// TIA Portal project "141db_PLcen hasera" (V15.1)

(* hardware
DEVICE "S7-1200 station_1"  S7-1200 Station
   slot 0: "Rack_0"  S7-1200 Rack  Rack  V1.0
   slot 1: "PLC_1"  CPU 1214C AC/DC/Rly  6ES7 214-1BG40-0XB0  V4.2
   slot 3: "AQ 1x12BIT_1"  AQ1 signal board  6ES7 232-4HA30-0XB0  V1.0
*)

// ===== PLC "PLC_1"  CPU 1214C AC/DC/Rly =====

VAR_GLOBAL   // PLC tag table "Tabla de variables estándar"
   "Etapa0" AT %M16.0 : Bool;
   "S1" AT %I1.0 : Bool;
   "CP" AT %I5.0 : Bool;
   "S2" AT %I2.0 : Bool;
   "P1" AT %Q1.0 : Bool;
   "S3" AT %I3.0 : Bool;
   "CG" AT %I6.0 : Bool;
   "Etapa1" AT %M16.1 : Bool;
   "Etapa2" AT %M16.2 : Bool;
   "Etapa3" AT %M16.3 : Bool;
   "Etapa4" AT %M16.4 : Bool;
   "Etapa5" AT %M16.5 : Bool;
   "Etapa6" AT %M16.6 : Bool;
   "P3" AT %Q3.0 : Bool;
   "P2" AT %Q2.0 : Bool;
END_VAR

// folder: System blocks/Program resources

DATA_BLOCK "Temporizador1"   // DB2
{ S7_Optimized_Access := 'TRUE' }
AUTHOR : Simatic
FAMILY : IEC
NAME : IEC_TMR
VERSION : 1.0
// stored: InstanceOfName IEC_TIMER
"IEC_TIMER"
BEGIN
END_DATA_BLOCK

DATA_BLOCK "Temporizador2"   // DB3
{ S7_Optimized_Access := 'TRUE' }
AUTHOR : Simatic
FAMILY : IEC
NAME : IEC_TMR
VERSION : 1.0
// stored: InstanceOfName IEC_TIMER
"IEC_TIMER"
BEGIN
END_DATA_BLOCK

DATA_BLOCK "Temporizador4"   // DB4
{ S7_Optimized_Access := 'TRUE' }
AUTHOR : Simatic
FAMILY : IEC
NAME : IEC_TMR
VERSION : 1.0
// stored: InstanceOfName IEC_TIMER
"IEC_TIMER"
BEGIN
END_DATA_BLOCK

// folder: (top level)

ORGANIZATION_BLOCK "Main"   // OB1, LAD, ProgramCycle
TITLE = "Main Program Sweep (Cycle)"
{ S7_Optimized_Access := 'TRUE' }
VERSION : 0.1
   VAR_INPUT
      Initial_Call : Bool;   // Initial call of this OB
      Remanence : Bool;   // =True, if remanent data are available
   END_VAR
   VAR_TEMP   // added for the SCL form of the ladder/FBD networks
      _w1 : Bool;
   END_VAR
BEGIN

REGION Network 1
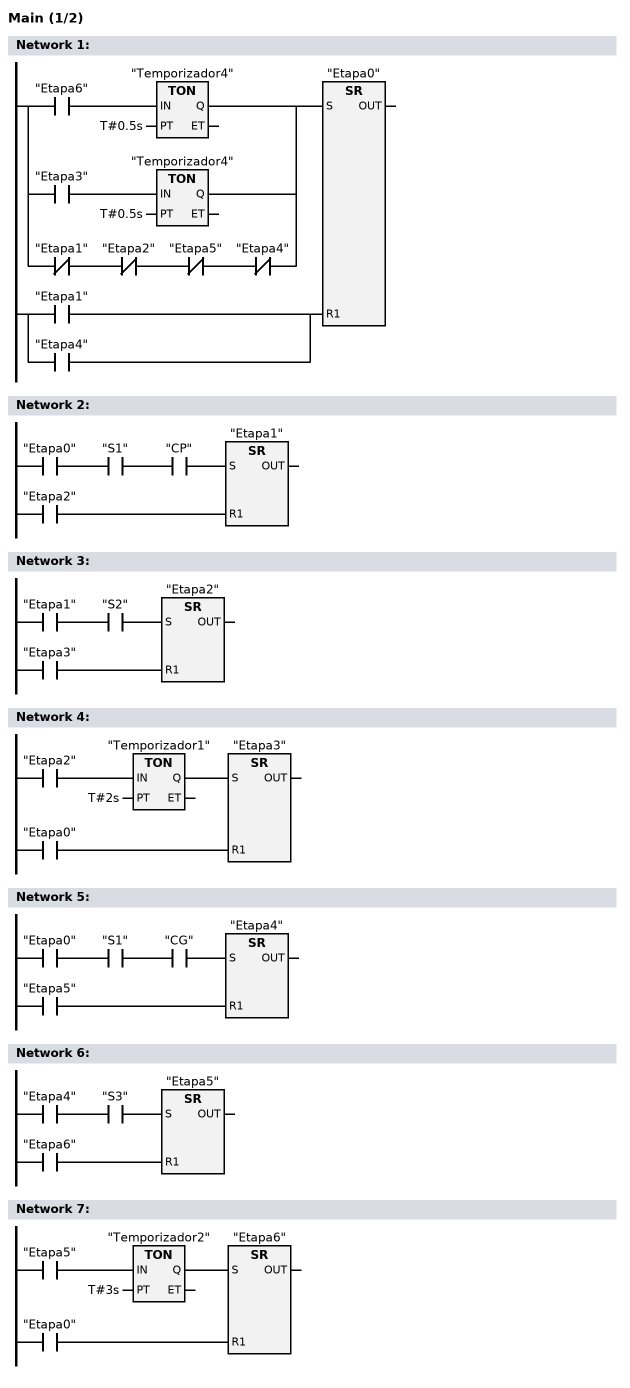
   "Temporizador4".TON(IN := "Etapa6", PT := T#0.5s);
   #_w1 := "Temporizador4".Q;
   "Temporizador4".TON(IN := "Etapa3", PT := T#0.5s);
   IF #_w1 OR "Temporizador4".Q OR (NOT "Etapa1" AND NOT "Etapa2" AND NOT "Etapa5" AND NOT "Etapa4") THEN
       "Etapa0" := TRUE;   // SR flip-flop
   END_IF;
   IF "Etapa1" OR "Etapa4" THEN "Etapa0" := FALSE; END_IF;
END_REGION

REGION Network 2
   RUNG wire#powerrail
      Contact( "Etapa0" )
      Contact( "S1" )
      Contact( "CP" )
      S_SR(operand := "Etapa1", r1 := wire#w1)
   END_RUNG
   RUNG wire#powerrail
      Contact( "Etapa2" )
   END_RUNG wire#w1
   // the same network as SCL:
   IF "Etapa0" AND "S1" AND "CP" THEN
       "Etapa1" := TRUE;   // SR flip-flop
   END_IF;
   IF "Etapa2" THEN "Etapa1" := FALSE; END_IF;
END_REGION

REGION Network 3
   RUNG wire#powerrail
      Contact( "Etapa1" )
      Contact( "S2" )
      S_SR(operand := "Etapa2", r1 := wire#w1)
   END_RUNG
   RUNG wire#powerrail
      Contact( "Etapa3" )
   END_RUNG wire#w1
   // the same network as SCL:
   IF "Etapa1" AND "S2" THEN
       "Etapa2" := TRUE;   // SR flip-flop
   END_IF;
   IF "Etapa3" THEN "Etapa2" := FALSE; END_IF;
END_REGION

REGION Network 4
   "Temporizador1".TON(IN := "Etapa2", PT := T#2s);
   IF "Temporizador1".Q THEN
       "Etapa3" := TRUE;   // SR flip-flop
   END_IF;
   IF "Etapa0" THEN "Etapa3" := FALSE; END_IF;
END_REGION

REGION Network 5
   RUNG wire#powerrail
      Contact( "Etapa0" )
      Contact( "S1" )
      Contact( "CG" )
      S_SR(operand := "Etapa4", r1 := wire#w1)
   END_RUNG
   RUNG wire#powerrail
      Contact( "Etapa5" )
   END_RUNG wire#w1
   // the same network as SCL:
   IF "Etapa0" AND "S1" AND "CG" THEN
       "Etapa4" := TRUE;   // SR flip-flop
   END_IF;
   IF "Etapa5" THEN "Etapa4" := FALSE; END_IF;
END_REGION

REGION Network 6
   RUNG wire#powerrail
      Contact( "Etapa4" )
      Contact( "S3" )
      S_SR(operand := "Etapa5", r1 := wire#w1)
   END_RUNG
   RUNG wire#powerrail
      Contact( "Etapa6" )
   END_RUNG wire#w1
   // the same network as SCL:
   IF "Etapa4" AND "S3" THEN
       "Etapa5" := TRUE;   // SR flip-flop
   END_IF;
   IF "Etapa6" THEN "Etapa5" := FALSE; END_IF;
END_REGION

REGION Network 7
   "Temporizador2".TON(IN := "Etapa5", PT := T#3s);
   IF "Temporizador2".Q THEN
       "Etapa6" := TRUE;   // SR flip-flop
   END_IF;
   IF "Etapa0" THEN "Etapa6" := FALSE; END_IF;
END_REGION

REGION Network 8
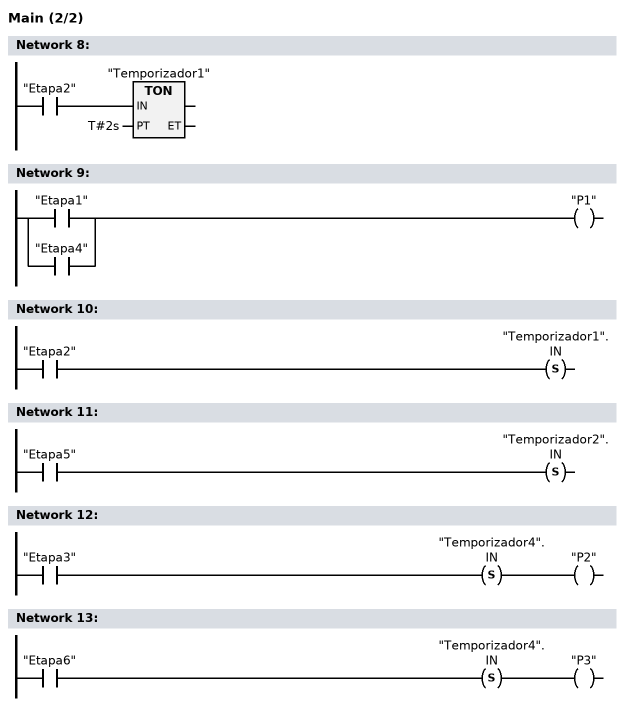
   "Temporizador1".TON(IN := "Etapa2", PT := T#2s);
END_REGION

REGION Network 9
   RUNG wire#powerrail
      Contact( "Etapa1" )
      wire#w1
      Coil( "P1" )
   END_RUNG
   RUNG wire#powerrail
      Contact( "Etapa4" )
   END_RUNG wire#w1
   // the same network as SCL:
   "P1" := "Etapa1" OR "Etapa4";
END_REGION

REGION Network 10
   RUNG wire#powerrail
      Contact( "Etapa2" )
      S_Coil( "Temporizador1".IN )
   END_RUNG
   // the same network as SCL:
   IF "Etapa2" THEN "Temporizador1".IN := TRUE; END_IF;
END_REGION

REGION Network 11
   RUNG wire#powerrail
      Contact( "Etapa5" )
      S_Coil( "Temporizador2".IN )
   END_RUNG
   // the same network as SCL:
   IF "Etapa5" THEN "Temporizador2".IN := TRUE; END_IF;
END_REGION

REGION Network 12
   RUNG wire#powerrail
      Contact( "Etapa3" )
      S_Coil( "Temporizador4".IN )
      Coil( "P2" )
   END_RUNG
   // the same network as SCL:
   IF "Etapa3" THEN "Temporizador4".IN := TRUE; END_IF;
   "P2" := "Etapa3";
END_REGION

REGION Network 13
   RUNG wire#powerrail
      Contact( "Etapa6" )
      S_Coil( "Temporizador4".IN )
      Coil( "P3" )
   END_RUNG
   // the same network as SCL:
   IF "Etapa6" THEN "Temporizador4".IN := TRUE; END_IF;
   "P3" := "Etapa6";
END_REGION
END_ORGANIZATION_BLOCK